{attribute 'qualified_only'}
{attribute 'strict'}
TYPE E_TIMER_STATE :
(
	STATE_TIMER_NONE				:= -1,
	STATE_TIMER_NOT_INIT,
	STATE_TIMER_INIT,
	STATE_TIMER_IDLE,
	STATE_TIMER_ARMED,
	STATE_TIMER_ACTIVE,
	STATE_TIMER_ERROR
);
END_TYPE

(* stored: Version 1.1.0.1, ProductVersion 3.1.4024.11
   DUT E_TIMER_STATE: Id {6e31b982-3c20-4935-bd49-546cc974fe82} *)
